SUBAPPLICATION SubApp_PC_B (* Geraet B (Station 12, 192.168.1.12): Toggle-Flipflop-Logik (AX_T_FF) und DigitalOutput_Q1 - 'SUB style', das Protokoll steckt im MyLib::sys-Composite (Toggle_RPC_FROM_Remote_QXA_OPC, wiederverwendet von Training_03), nicht in der Resource des Geraets - Toggle-alleine-Variante von Training_04/06, manuelle Verdrahtung (wie Training_04), gleiche OPC-UA-Adressen wie Training_03 *)
  (* Standard: 61499-2; Description: Copyright (c) 2026 Meisterschulen am Ostbahnhof This program and the accompanying materials are made available under the terms of the Eclipse Public License 2.0 which is available at https://www.eclipse.org/legal/epl-2.0/ SPDX-License-Identifier: EPL-2.0 *)
  (* Version 1.0, 2026-09-04, Franz Höpfinger, Meisterschulen am Ostbahnhof, initial API and implementation and/or initial documentation *)
  PACKAGE subapp::Training_08_OPC_UA_RES;
  IMPORT logiBUS::io::DQ::logiBUS_DO::Output_Q1;
  IMPORT VV::const::OPC_UA::myOpcUaAddresses::FF1_TRIGGER_LOCAL_METHOD;
  IMPORT VV::const::OPC_UA::myOpcUaAddresses::FF1_STATE_REMOTE_WRITE;
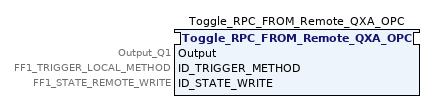
  SUBAPPS
    Toggle_RPC_FROM_Remote_QXA_OPC : MyLib::sys::Toggle_RPC_FROM_Remote_QXA_OPC(Output := Output_Q1, ID_TRIGGER_METHOD := FF1_TRIGGER_LOCAL_METHOD, ID_STATE_WRITE := FF1_STATE_REMOTE_WRITE);
  END_SUBAPPS
END_SUBAPPLICATION
